(* IEC 61131-3 sources: SRCI/RobotLibrary/Library/POUs/General/MC_ReadServerLog_ToDo, 1 file *)

(* ---- MC_ReadServerLog.st ---- *)
FUNCTION_BLOCK MC_ReadServerLog EXTENDS RobotLibraryBaseFB
VAR
END_VAR

END_FUNCTION_BLOCK

METHOD FB_init : BOOL
VAR_INPUT
  /// if TRUE, the retain variables are initialized (warm start / cold start)
  bInitRetains : BOOL;
  /// if TRUE, the instance afterwards gets moved into the copy code (online change)
  bInCopyCode  : BOOL;
END_VAR

  MyType := 'MC_ReadServerLogFB';

  ExecMode := ExecutionMode.PARALLEL;
  Priority := PriorityLevel.NORMAL;

END_METHOD
